// TIA Portal V15.1 export
// export: Created 2026-01-09T13:45:11.8507823Z, ExportSetting WithDefaults, WithReadOnly, DisplayName Totally Integrated Automation Portal, DisplayVersion V15.1 Update 8, DisplayName TIA Portal Openness, DisplayVersion V15.1 Update 8, DisplayName STEP 7 Professional, DisplayVersion V15.1 Update 8, DisplayName WinCC Advanced, DisplayVersion V15.1 Update 8
DATA_BLOCK "C#8_RD_REPORT"   // DB8
{ S7_Optimized_Access := 'FALSE' }
VERSION : 0.1
// stored: AutoNumber false, CodeModifiedDate 2024-09-25T16:49:35.7764199Z, CompileDate 2025-08-30T17:40:31.7117876Z, CreationDate 2024-10-12T12:36:08.0193576Z, DBAccessibleFromOPCUA true, InterfaceModifiedDate 2024-09-25T16:49:35.7764199Z, IsConsistent true, IsKnowHowProtected false, IsOnlyStoredInLoadMemory false, IsPLCDB false, IsWriteProtectedInAS false, ModifiedDate 2024-10-13T07:15:20.7288707Z, ParameterModified 2024-09-25T16:49:35.7764199Z, StructureModified 2024-09-25T16:49:35.7764199Z
   VAR
      SAVE_REPORT : Bool;   // Lưu dữ liệu trộn
      SAVE_REPORT_1 : Bool;
      SAVE_REPORT_2 : Bool;
      SAVE_REPORT_3 : Bool;
      SAVE_REPORT_4 : Bool;
      SAVE_REPORT_5 : Bool;
      SAVE_REPORT_6 : Bool;
      SAVE_REPORT_7 : Bool;
      SAVE_REPORT_8 : Bool;
      SAVE_REPORT_9 : Bool;
      SAVE_REPORT_10 : Bool;
      SAVE_REPORT_11 : Bool;
      SAVE_REPORT_12 : Bool;
      SAVE_REPORT_13 : Bool;
      SAVE_REPORT_14 : Bool;
      SAVE_REPORT_15 : Bool;
      SAVE_REPORT_16 : Bool;
      PV_AGG1 : Real;   // Thực cân Cốt liệu 1
      PVM_AGG1 : Real;   // Cân tay Cốt liệu 1
      PV_AGG2 : Real;   // Thực cân Cốt liệu 2
      PVM_AGG2 : Real;   // Cân tay Cốt liệu 2
      PV_AGG3 : Real;   // Thực cân Cốt liệu 3
      PVM_AGG3 : Real;   // Cân tay Cốt liệu 3
      PV_AGG4 : Real;   // Thực cân Cốt liệu 4
      PVM_AGG4 : Real;   // Cân tay Cốt liệu 4
      PV_AGG5 : Real;   // Thực cân Cốt liệu 5
      PVM_AGG5 : Real;   // Cân tay Cốt liệu 5
      TEMP_TS : Real;   // Nhiệt độ tang sấy
      TEMP_AG : Real;   // Nhiệt độ cốt liệu
      PV_FD1 : Real;   // Thực cân F/D 1
      PVM_FD1 : Real;   // Cân tay F/D 1
      PV_AP1 : Real;   // Thực cân Nhựa 1
      PVM_AP1 : Real;   // Cân tay Nhựa 1
      TEMP_AP : Real;   // Nhiệt độ nhựa
      PV_SB1 : Real;   // Thực cân SBS 1
      PVM_SB1 : Real;   // Cân tay SBS 1
   END_VAR
BEGIN
END_DATA_BLOCK
